// TIA Portal V20 export
TYPE "LER_typeAlignMoveCalibrationCommands"
// stored: Access Published
   STRUCT
      stepStart : Bool;
      stepStop : Bool;
      errorAck : Bool;
      Apply : Bool;
      MovePos1 : Bool;
      MovePos2 : Bool;
      MovePos3 : Bool;
      MovePos4 : Bool;
      MovePos5 : Bool;
      MovePos6 : Bool;
      MovePos7 : Bool;
      MovePos8 : Bool;
      MovePos9 : Bool;
   END_STRUCT;
END_TYPE
